ABB RAPID module: P2545L1ESegmentOrg.mod

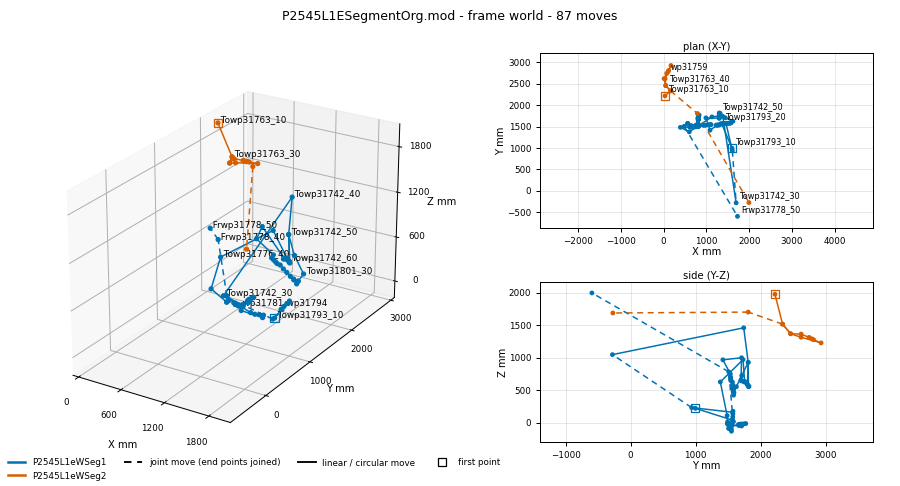
[picture p0: tool path of P2545L1ESegmentOrg.mod in frame world, 87 of 89 moves have a stored position in this frame; points joined in program order, loops and branches not executed]
%%%
  VERSION:1
  LANGUAGE:ENGLISH
%%%

MODULE P2545L1ESegment
!# Process Simulate on eMServer 14 to ABB Rapid Volvo download
!# ------------------------------------------------
!# CREATED   : 26/04/2018 14:09:44 by yogesha
!# CELL      : 2V3 Enginecase_V1
!# ROBOT     : AR21_IRB6700_220-265_SW_IRC5_Grey
!# PROGRAM   : P2545L1ESegment
!# VOLP      : Abb-Rapid-Volvo 3.14.1
!# RCS       : 6.04.irc5
!# CONTROLLER: 6.0 RW6


!# ----------------------------------------------
!# ------ ROBTARGET
!# ----------------------------------------------
  LOCAL CONST robtarget Towp31793_10:=[[4045.55,-245.18,1773.35],[0.031229,0.227881,0.973063,0.015622],[-1,0,-1,0],[9e+09,250,9e+09,9e+09,9e+09,9e+09]];
  LOCAL CONST robtarget Towp31793_20:=[[3464.22,18.06,1738.48],[0.0312267,0.227864,0.973067,0.0156211],[0,0,-1,0],[9E+09,250,9E+09,9E+09,9E+09,9E+09]];
  LOCAL CONST robtarget wp31793:=[[3459.52,28.59,1728.27],[0.0311732,0.227874,0.973066,0.0155927],[0,0,-1,0],[9E+09,24.9994,9E+09,9E+09,9E+09,9E+09]];
  LOCAL CONST robtarget wp31794:=[[3457.21,-31.09,1727.85],[0.0295957,0.184936,0.982299,0.00348625],[0,0,-1,0],[9E+09,25.0015,9E+09,9E+09,9E+09,9E+09]];
  LOCAL CONST robtarget wp31795:=[[3457.59,-92.13,1727.10],[0.0256679,0.112505,0.99332,0.000286719],[-1,1,-1,0],[9E+09,24.9989,9E+09,9E+09,9E+09,9E+09]];
  LOCAL CONST robtarget wp31796:=[[3459.26,-148.29,1728.07],[0.024545,0.091993,0.995457,-0.000992369],[-1,1,-1,0],[9E+09,24.9989,9E+09,9E+09,9E+09,9E+09]];
  LOCAL CONST robtarget Towp31742_10:=[[3464.44,-137.28,1737.71],[0.024542,0.091977,0.995458,-0.00102],[-1,1,-1,0],[9e+09,250,9e+09,9e+09,9e+09,9e+09]];
  LOCAL CONST robtarget Towp31742_20:=[[4102.65,-256.3,1769.61],[0.024542,0.091977,0.995458,-0.00102],[-1,0,-1,0],[9e+09,250,9e+09,9e+09,9e+09,9e+09]];
  LOCAL CONST robtarget Towp31742_30:=[[5323.84,-882.05,1248.86],[0.389563,-0.196475,-0.871387,-0.224327],[-1,0,-1,0],[9e+09,250,9e+09,9e+09,9e+09,9e+09]];
  LOCAL CONST robtarget Towp31742_40:=[[3288.74,-1093.58,858.48],[0.205443,-0.383752,-0.808886,-0.395262],[0,-1,0,0],[9E+09,200,9E+09,9E+09,9E+09,9E+09]];
  LOCAL CONST robtarget Towp31742_50:=[[3214.45,-634.81,1138.27],[0.192085,-0.483988,-0.79404,-0.313623],[0,-1,0,0],[9e+09,200,9e+09,9e+09,9e+09,9e+09]];
  LOCAL CONST robtarget Towp31742_60:=[[3228.3,-383.45,1373.91],[0.192085,-0.483988,-0.79404,-0.313623],[0,-1,0,0],[9e+09,200,9e+09,9e+09,9e+09,9e+09]];
  LOCAL CONST robtarget wp31742:=[[3218.38,-372.34,1363.36],[0.19209,-0.483981,-0.794042,-0.313625],[0,-1,0,0],[9E+09,25,9E+09,9E+09,9E+09,9E+09]];
  LOCAL CONST robtarget wp31743:=[[3202.14,-353.55,1377.18],[0.126687,-0.453575,-0.849352,-0.238374],[0,-1,0,0],[9E+09,25,9E+09,9E+09,9E+09,9E+09]];
  LOCAL CONST robtarget Towp31801_10:=[[3211.68,-359.85,1390.85],[0.126681,-0.453575,-0.849353,-0.238372],[0,-1,0,0],[9e+09,100,9e+09,9e+09,9e+09,9e+09]];
  LOCAL CONST robtarget Towp31801_20:=[[3214.45,-634.81,1138.27],[0.192085,-0.483988,-0.79404,-0.313623],[0,-1,0,0],[9e+09,200,9e+09,9e+09,9e+09,9e+09]];
  LOCAL CONST robtarget Towp31801_50:=[[3324.02,-564.37,1372.17],[0.253684,-0.525737,-0.694294,-0.420952],[0,-1,0,0],[9E+09,252.271,9E+09,9E+09,9E+09,9E+09]];
  LOCAL CONST robtarget Towp31801_30:=[[3418.53,-543.62,1612.1],[0.303641,-0.551478,-0.586786,-0.509271],[0,-1,1,0],[9e+09,300,9e+09,9e+09,9e+09,9e+09]];
  LOCAL CONST robtarget Towp31801_40:=[[3453.83,-438.28,1630.24],[0.30364,-0.551504,-0.586755,-0.509279],[0,-2,1,0],[9e+09,250,9e+09,9e+09,9e+09,9e+09]];
  LOCAL CONST robtarget wp31801:=[[3456.41,-397.01,1641.04],[0.303642,-0.551506,-0.586753,-0.509277],[0,-2,1,0],[9E+09,24.9995,9E+09,9E+09,9E+09,9E+09]];
  LOCAL CONST robtarget Towp31802_10:=[[3453.84,-438.28,1630.24],[0.30364,-0.551504,-0.586755,-0.509279],[0,-2,1,0],[9e+09,250,9e+09,9e+09,9e+09,9e+09]];
  LOCAL CONST robtarget Towp31802_20:=[[3460.41,-415.7,1573.72],[0.426749,-0.48377,-0.53862,-0.541977],[1,-2,1,0],[9e+09,250,9e+09,9e+09,9e+09,9e+09]];
  LOCAL CONST robtarget wp31802:=[[3457.06,-406.72,1584.59],[0.426746,-0.48378,-0.538616,-0.541976],[0,-2,1,0],[9E+09,25,9E+09,9E+09,9E+09,9E+09]];
  LOCAL CONST robtarget wp31803:=[[3459.02,-406.42,1523.09],[0.43668,-0.46746,-0.526416,-0.560069],[1,-2,1,0],[9E+09,25.0005,9E+09,9E+09,9E+09,9E+09]];
  LOCAL CONST robtarget wp31804:=[[3459.21,-407.58,1459.46],[0.445685,-0.447678,-0.547002,-0.549307],[1,-2,1,0],[9E+09,25,9E+09,9E+09,9E+09,9E+09]];
  LOCAL CONST robtarget wp31805:=[[3459.16,-405.57,1400.86],[0.452433,-0.455769,-0.540253,-0.543788],[1,-2,1,0],[9E+09,25,9E+09,9E+09,9E+09,9E+09]];
  LOCAL CONST robtarget wp31806:=[[3458.52,-409.86,1340.90],[0.439789,-0.439763,-0.5538,-0.553624],[1,-2,1,0],[9E+09,25,9E+09,9E+09,9E+09,9E+09]];
  LOCAL CONST robtarget wp400071:=[[3480.23,-407.44,1303.25],[0.415408,-0.44219,-0.578614,-0.545078],[1,-2,1,0],[9E+09,24.9993,9E+09,9E+09,9E+09,9E+09]];
  LOCAL CONST robtarget wp31807:=[[3480.96,-408.30,1277.13],[0.429146,-0.4291,-0.56212,-0.561897],[1,-2,1,0],[9E+09,25,9E+09,9E+09,9E+09,9E+09]];
  LOCAL CONST robtarget wp31808:=[[3479.48,-405.77,1244.18],[0.421356,-0.421308,-0.567923,-0.567823],[1,-2,1,0],[9E+09,25.0005,9E+09,9E+09,9E+09,9E+09]];
  LOCAL CONST robtarget wp31809:=[[3480.49,-404.93,1208.70],[0.421373,-0.421325,-0.56793,-0.56779],[1,-2,1,0],[9E+09,25,9E+09,9E+09,9E+09,9E+09]];
  LOCAL CONST robtarget Towp31738_10:=[[3484.07,-455.96,1198.82],[0.421374,-0.421319,-0.56794,-0.567784],[1,-2,1,0],[9e+09,200,9e+09,9e+09,9e+09,9e+09]];
  LOCAL CONST robtarget Towp31738_20:=[[3587.28,-510.98,927.08],[0.421374,-0.421319,-0.56794,-0.567784],[1,-2,1,0],[9e+09,200,9e+09,9e+09,9e+09,9e+09]];
  LOCAL CONST robtarget Towp31738_30:=[[3293.19,-486.33,848.58],[0.312249,-0.509804,-0.662688,-0.45105],[1,-1,1,0],[9E+09,100,9E+09,9E+09,9E+09,9E+09]];
  LOCAL CONST robtarget Towp31738_40:=[[3325.04,-426.92,1307.08],[0.481537,-0.548607,-0.510598,-0.454358],[1,-1,1,0],[9e+09,100,9e+09,9e+09,9e+09,9e+09]];
  LOCAL CONST robtarget wp31738:=[[3321.4,-408.44,1309.01],[0.481539,-0.548608,-0.510599,-0.454355],[1,-1,1,0],[9E+09,25,9E+09,9E+09,9E+09,9E+09]];
  LOCAL CONST robtarget wp31739:=[[3289.73,-404.44,1319.17],[0.411306,-0.529111,-0.571082,-0.474061],[1,-1,1,0],[9E+09,25,9E+09,9E+09,9E+09,9E+09]];
  LOCAL CONST robtarget wp31740:=[[3264.45,-398.53,1332.57],[0.350381,-0.565629,-0.615727,-0.42211],[0,-1,1,0],[9E+09,25,9E+09,9E+09,9E+09,9E+09]];
  LOCAL CONST robtarget Towp31776_10:=[[3270.4,-418.62,1333.94],[0.350381,-0.565628,-0.615725,-0.422114],[0,-1,1,0],[9e+09,100,9e+09,9e+09,9e+09,9e+09]];
  LOCAL CONST robtarget Towp31776_20:=[[3280.95,-555.22,975.55],[0.31225,-0.509807,-0.662682,-0.451053],[0,-1,1,0],[9e+09,200,9e+09,9e+09,9e+09,9e+09]];
  LOCAL CONST robtarget Towp31776_40:=[[3591.17,61.90,770.34],[0.307479,0.489827,-0.385208,0.719125],[1,-1,-1,0],[9E+09,200,9E+09,9E+09,9E+09,9E+09]];
  LOCAL CONST robtarget Towp31776_50:=[[3471.36,587.04,948.32],[0.504101,0.53927,-0.460831,0.492651],[1,-1,-1,0],[9E+09,200,9E+09,9E+09,9E+09,9E+09]];
  LOCAL CONST robtarget Towp31776_60:=[[3480,543.53,1199.86],[0.528139,0.542024,-0.467947,0.456404],[1,-1,-1,0],[9e+09,200,9e+09,9e+09,9e+09,9e+09]];
  LOCAL CONST robtarget wp31776:=[[3483.05,500.39,1205.78],[0.528141,0.542017,-0.46796,0.456396],[1,-1,-1,0],[9E+09,24.9917,9E+09,9E+09,9E+09,9E+09]];
  LOCAL CONST robtarget Towp31780_10:=[[3480,543.52,1199.86],[0.528138,0.542024,-0.467947,0.456404],[1,-1,-1,0],[9e+09,200,9e+09,9e+09,9e+09,9e+09]];
  LOCAL CONST robtarget Towp31780_20:=[[3390.65,544.94,1142.27],[0.528139,0.542024,-0.467946,0.456404],[1,-1,-1,0],[9e+09,200,9e+09,9e+09,9e+09,9e+09]];
  LOCAL CONST robtarget Towp31780_30:=[[3451.46,472,1330.74],[0.485437,0.649543,-0.468784,0.350265],[1,-1,-1,0],[9e+09,150,9e+09,9e+09,9e+09,9e+09]];
  LOCAL CONST robtarget wp31780:=[[3482.98,440.49,1321.01],[0.48544,0.649557,-0.468776,0.350246],[1,-1,-1,0],[9E+09,25,9E+09,9E+09,9E+09,9E+09]];
  LOCAL CONST robtarget wp31781:=[[3482.35,428.05,1352.01],[0.442766,0.654013,-0.507582,0.344363],[1,-1,-1,0],[9E+09,25.0005,9E+09,9E+09,9E+09,9E+09]];
  LOCAL CONST robtarget wp31785:=[[3464.69,396.47,1497.30],[0.470942,0.633397,-0.47932,0.383763],[1,-1,-1,0],[9E+09,25,9E+09,9E+09,9E+09,9E+09]];
  LOCAL CONST robtarget wp31786:=[[3461.70,368.27,1546.79],[0.379891,0.694641,-0.526925,0.309043],[1,-1,-1,0],[9E+09,25.0005,9E+09,9E+09,9E+09,9E+09]];
  LOCAL CONST robtarget wp31787:=[[3459.50,323.86,1589.21],[0.24633,0.70303,-0.621694,0.242006],[1,-1,-1,0],[9E+09,25.0005,9E+09,9E+09,9E+09,9E+09]];
  LOCAL CONST robtarget wp31788:=[[3459.95,282.60,1629.14],[0.353136,0.765889,-0.477535,0.246312],[1,-1,-1,0],[9E+09,24.9995,9E+09,9E+09,9E+09,9E+09]];
  LOCAL CONST robtarget Towp31782_10:=[[3455.66,320.67,1642.93],[0.353143,0.76587,-0.477559,0.246314],[1,-1,-1,0],[9e+09,100,9e+09,9e+09,9e+09,9e+09]];
  LOCAL CONST robtarget Towp31782_20:=[[3479.58,469.31,1398.3],[0.371118,0.727003,-0.513868,0.263966],[1,-1,-1,0],[9e+09,200,9e+09,9e+09,9e+09,9e+09]];
  LOCAL CONST robtarget wp31782:=[[3480.26,418.82,1363.79],[0.371131,0.726978,-0.513897,0.263958],[1,-1,-1,0],[9E+09,24.9974,9E+09,9E+09,9E+09,9E+09]];
  LOCAL CONST robtarget wp31775:=[[3460.80,422.79,1361.94],[0.369179,0.711005,-0.532671,0.272839],[1,-1,-1,0],[9E+09,24.9878,9E+09,9E+09,9E+09,9E+09]];
  LOCAL CONST robtarget wp31774:=[[3430.48,422.82,1360.70],[0.3679,0.715304,-0.528284,0.271855],[1,-1,-1,0],[9E+09,25,9E+09,9E+09,9E+09,9E+09]];
  LOCAL CONST robtarget Towp31767_10:=[[3431.36,435.91,1374.3],[0.36792,0.715269,-0.52832,0.271852],[1,-1,-1,0],[9e+09,75,9e+09,9e+09,9e+09,9e+09]];
  LOCAL CONST robtarget Towp31767_20:=[[3322.44,425.06,1380.62],[0.266606,0.650081,-0.667266,0.247126],[1,-1,-1,0],[9E+09,49.4176,9E+09,9E+09,9E+09,9E+09]];
  LOCAL CONST robtarget wp31767:=[[3217.64,388.64,1378.16],[0.161313,0.567008,-0.778505,0.21543],[1,-1,0,0],[9E+09,24.9979,9E+09,9E+09,9E+09,9E+09]];
  LOCAL CONST robtarget wp31768:=[[3241.82,402.64,1368.34],[0.265979,0.686435,-0.632244,0.241516],[1,-1,-1,0],[9E+09,25.0005,9E+09,9E+09,9E+09,9E+09]];
  LOCAL CONST robtarget wp31771:=[[3328.78,419.32,1363.33],[0.343843,0.752013,-0.470483,0.308051],[1,-1,-1,0],[9E+09,25,9E+09,9E+09,9E+09,9E+09]];
  LOCAL CONST robtarget wp31770:=[[3302.45,416.94,1357.38],[0.285253,0.752472,-0.498291,0.32268],[1,-1,-1,0],[9E+09,25,9E+09,9E+09,9E+09,9E+09]];
  LOCAL CONST robtarget wp31769:=[[3275.95,412.76,1358.82],[0.281989,0.697675,-0.612726,0.241452],[1,-1,-1,0],[9E+09,25,9E+09,9E+09,9E+09,9E+09]];
  LOCAL CONST robtarget Towp31779_10:=[[3279.73,435.49,1380.14],[0.281999,0.69766,-0.612741,0.241446],[1,-1,-1,0],[9e+09,75,9e+09,9e+09,9e+09,9e+09]];
  LOCAL CONST robtarget Towp31779_20:=[[3480.1,470.7,1295.95],[0.363356,0.754516,-0.492864,0.236144],[1,-1,-1,0],[9e+09,25,9e+09,9e+09,9e+09,9e+09]];
  LOCAL CONST robtarget wp31779:=[[3482.68,451.68,1288.55],[0.363388,0.754466,-0.492923,0.23613],[1,-1,-1,0],[9E+09,25,9E+09,9E+09,9E+09,9E+09]];
  LOCAL CONST robtarget wp31778:=[[3481.75,469.66,1267.37],[0.319477,0.752877,-0.529636,0.224937],[1,-1,-1,0],[9E+09,25.0005,9E+09,9E+09,9E+09,9E+09]];
  LOCAL CONST robtarget Frwp31778_10:=[[3480.1,470.71,1295.94],[0.363356,0.754516,-0.492864,0.236144],[1,-1,-1,0],[9e+09,75,9e+09,9e+09,9e+09,9e+09]];
  LOCAL CONST robtarget Frwp31778_20:=[[3451.42,471.98,1330.73],[0.550376,0.597256,-0.47701,0.335906],[1,-1,-1,0],[9E+09,75,9E+09,9E+09,9E+09,9E+09]];
  LOCAL CONST robtarget Frwp31778_30:=[[3390.65,544.94,1142.27],[0.528139,0.542024,-0.467946,0.456404],[1,-1,-1,0],[9e+09,100,9e+09,9e+09,9e+09,9e+09]];
  LOCAL CONST robtarget Frwp31778_40:=[[3452.82,11.54,588.04],[0.294229,0.459328,-0.391939,0.740831],[1,-1,-1,0],[9E+09,50,9E+09,9E+09,9E+09,9E+09]];
  LOCAL CONST robtarget Frwp31778_50:=[[6079.26,2565.85,1512.62],[0.516372,-0.844715,-0.107098,-0.091356],[0,-1,-2,0],[9e+09,50,9e+09,9e+09,9e+09,9e+09]];
  LOCAL CONST robtarget Towp31763_10:=[[3347.95,834.06,944.48],[0.127354,-0.51805,0.839702,0.101518],[0,0,-2,0],[9E+09,242,9E+09,9E+09,9E+09,9E+09]];
  LOCAL CONST robtarget Towp31763_30:=[[3426.57,520.60,1315.50],[0.184335,-0.578608,0.784931,-0.122949],[0,0,-2,0],[9E+09,242.273,9E+09,9E+09,9E+09,9E+09]];
  LOCAL CONST robtarget Towp31763_40:=[[3274.99,407.18,1434.32],[0.0363429,-0.545988,0.805467,-0.227595],[0,0,-2,0],[9E+09,242.273,9E+09,9E+09,9E+09,9E+09]];
  LOCAL CONST robtarget wp31763:=[[3171.50,283.07,1395.44],[6.03512E-05,0.582137,-0.813091,0.000137078],[1,0,-2,0],[9E+09,24.9948,9E+09,9E+09,9E+09,9E+09]];
  LOCAL CONST robtarget wp31759:=[[3176.67,136.97,1394.83],[0.0193566,-0.592124,0.805535,-0.0112687],[1,0,-2,0],[9E+09,24.9966,9E+09,9E+09,9E+09,9E+09]];
  LOCAL CONST robtarget wp31757:=[[3187.80,79.83,1395.86],[0.00985179,-0.606855,0.79473,-0.00582832],[1,0,-2,0],[9E+09,24.9978,9E+09,9E+09,9E+09,9E+09]];
  LOCAL CONST robtarget wp31756:=[[3187.98,48.79,1398.52],[8.77831E-06,0.626617,-0.779328,5.44794E-05],[1,-1,-2,0],[9E+09,25,9E+09,9E+09,9E+09,9E+09]];
  LOCAL CONST robtarget wp31752:=[[3189.26,-88.41,1398.85],[4.25555E-05,0.644101,-0.76494,0.000169744],[1,-1,-2,0],[9E+09,24.9996,9E+09,9E+09,9E+09,9E+09]];
  LOCAL CONST robtarget Frwp31752_10:=[[3195.54,257.28,1437.13],[0.0242655,-0.583135,0.797612,-0.152251],[0,0,-2,0],[9E+09,169.434,9E+09,9E+09,9E+09,9E+09]];
  LOCAL CONST robtarget Frwp31752_20:=[[3275.00,407.18,1434.32],[0.0363422,-0.54599,0.805466,-0.227593],[0,0,-2,0],[9E+09,242.273,9E+09,9E+09,9E+09,9E+09]];
  LOCAL CONST robtarget Frwp31752_30:=[[3426.57,520.60,1315.50],[0.184334,-0.578607,0.784932,-0.122949],[0,0,-2,0],[9E+09,242.273,9E+09,9E+09,9E+09,9E+09]];
  LOCAL CONST robtarget Frwp31752_50:=[[4215.11,789.08,1199.66],[0.410337,-0.682659,0.516184,-0.314887],[0,0,-2,0],[9e+09,10,9e+09,9e+09,9e+09,9e+09]];
  LOCAL CONST robtarget Frwp31752_60:=[[6189.98,2078.46,1654.43],[0.626282,-0.760131,-0.076663,-0.155225],[0,0,-2,0],[9e+09,10,9e+09,9e+09,9e+09,9e+09]];


!# -----------------------------------------------
!# ------ SPOT DATA
!# -----------------------------------------------
  LOCAL PERS spotdata Sd_wp31793:=[3179320,1,1,1,1,-1];
  LOCAL PERS spotdata Sd_wp31794:=[3179420,1,1,1,1,-1];
  LOCAL PERS spotdata Sd_wp31795:=[3179520,1,1,1,1,-1];
  LOCAL PERS spotdata Sd_wp31796:=[3179620,1,1,1,1,-1];
  LOCAL PERS spotdata Sd_wp31742:=[3174220,1,1,1,1,-1];
  LOCAL PERS spotdata Sd_wp31743:=[3174320,1,1,1,1,-1];
  LOCAL PERS spotdata Sd_wp31801:=[3180120,1,1,1,1,-1];
  LOCAL PERS spotdata Sd_wp31802:=[3180220,1,1,1,1,-1];
  LOCAL PERS spotdata Sd_wp31803:=[3180320,1,1,1,1,-1];
  LOCAL PERS spotdata Sd_wp31804:=[3180420,1,1,1,1,-1];
  LOCAL PERS spotdata Sd_wp31805:=[3180520,1,1,1,1,-1];
  LOCAL PERS spotdata Sd_wp31806:=[3180620,1,1,1,1,-1];
  LOCAL PERS spotdata Sd_wp400071:=[4007120,1,1,1,1,-1];
  LOCAL PERS spotdata Sd_wp31807:=[3180720,1,1,1,1,-1];
  LOCAL PERS spotdata Sd_wp31808:=[3180820,1,1,1,1,-1];
  LOCAL PERS spotdata Sd_wp31809:=[3180920,1,1,1,1,-1];
  LOCAL PERS spotdata Sd_wp31738:=[3173820,1,1,1,1,-1];
  LOCAL PERS spotdata Sd_wp31739:=[3173920,1,1,1,1,-1];
  LOCAL PERS spotdata Sd_wp31740:=[3174020,1,1,1,1,-1];
  LOCAL PERS spotdata Sd_wp31780:=[3178020,1,1,1,1,-1];
  LOCAL PERS spotdata Sd_wp31781:=[3178120,1,1,1,1,-1];
  LOCAL PERS spotdata Sd_wp31785:=[3178520,1,1,1,1,-1];
  LOCAL PERS spotdata Sd_wp31786:=[3178620,1,1,1,1,-1];
  LOCAL PERS spotdata Sd_wp31787:=[3178720,1,1,1,1,-1];
  LOCAL PERS spotdata Sd_wp31788:=[3178820,1,1,1,1,-1];
  LOCAL PERS spotdata Sd_wp31782:=[3178220,1,1,1,1,-1];
  LOCAL PERS spotdata Sd_wp31775:=[3177520,1,1,1,1,-1];
  LOCAL PERS spotdata Sd_wp31774:=[3177420,1,1,1,1,-1];
  LOCAL PERS spotdata Sd_wp31767:=[3176720,1,1,1,1,-1];
  LOCAL PERS spotdata Sd_wp31768:=[3176820,1,1,1,1,-1];
  LOCAL PERS spotdata Sd_wp31771:=[3177120,1,1,1,1,-1];
  LOCAL PERS spotdata Sd_wp31770:=[3177020,1,1,1,1,-1];
  LOCAL PERS spotdata Sd_wp31769:=[3176920,1,1,1,1,-1];
  LOCAL PERS spotdata Sd_wp31779:=[3177920,1,1,1,1,-1];
  LOCAL PERS spotdata Sd_wp31778:=[3177820,1,1,1,1,-1];
  LOCAL PERS spotdata Sd_wp31763:=[3176320,1,1,1,1,-1];
  LOCAL PERS spotdata Sd_wp31759:=[3175920,1,1,1,1,-1];
  LOCAL PERS spotdata Sd_wp31757:=[3175720,1,1,1,1,-1];
  LOCAL PERS spotdata Sd_wp31756:=[3175620,1,1,1,1,-1];
  LOCAL PERS spotdata Sd_wp31752:=[3175220,1,1,1,1,-1];
  LOCAL PERS spotdata Sd_wp31776:=[3177620,1,1,1,1,-1];

!# -----------------------------------------------
!# ------ WOBJ DATA
!# -----------------------------------------------
  PERS wobjdata wFM24_CabframeUQ53:=[FALSE,TRUE,"""",[[-210.08,4920.13,1168.24],[-0.310764,0.6630223,-0.6166411,0.2891035]],[[0,0,0],[1,0,0,0]]];
  PERS wobjdata wFM24_CabframeUQ54:=[FALSE,TRUE,"""",[[-212.9,4917.65,1167.66],[-0.3109636,0.6634134,-0.6162131,0.2889042]],[[0,0,0],[1,0,0,0]]];
  PERS wobjdata wFM24_Cabframe:=[FALSE,TRUE,"""",[[-210.08,4920.13,1168.24],[-0.310764,0.663022,-0.616641,0.289104]],[[0,0,0],[1,0,0,0]]];
  PERS wobjdata wFM24_CabframeGrip:=[FALSE,TRUE,"""",[[-2504.52,4649.77,2641.4],[0.1735002,0.9601499,-0.2131685,-0.0506865]],[[0,0,0],[1,0,0,0]]];




  PROC P2545L1eWSeg1()
     MoveAbsJ HomeXQ11Gun,v2500,fine,XQ11GunTCP;
     MoveL Towp31793_10,v2500,z200,XQ11GunTCP\Wobj:=wFM24_Cabframe;
     MoveL Towp31793_20,v2500,z50,XQ11GunTCP\Wobj:=wFM24_Cabframe;
     SpotL wp31793, v2500, XQ11Gun\GunD:=XQ11GunData, Sd_wp31793, XQ11GunTCP\WObj:=wFM24_Cabframe;
     SpotL wp31794, v2500, XQ11Gun\GunD:=XQ11GunData, Sd_wp31794, XQ11GunTCP\WObj:=wFM24_Cabframe;
     SpotL wp31795, v2500, XQ11Gun\GunD:=XQ11GunData, Sd_wp31795, XQ11GunTCP\WObj:=wFM24_Cabframe;
     SpotL wp31796, v2500, XQ11Gun\GunD:=XQ11GunData, Sd_wp31796, XQ11GunTCP\WObj:=wFM24_Cabframe;
     MoveL Towp31742_10,v2500,z200,XQ11GunTCP\Wobj:=wFM24_Cabframe;
     MoveL Towp31742_20,v2500,z200,XQ11GunTCP\Wobj:=wFM24_Cabframe;
     MoveJ Towp31742_30,v2500,z200,XQ11GunTCP\Wobj:=wFM24_Cabframe;
     MoveL Towp31742_40,v2500,z200,XQ11GunTCP\Wobj:=wFM24_Cabframe;
     MoveL Towp31742_50,v2500,z50,XQ11GunTCP\Wobj:=wFM24_Cabframe;
     MoveL Towp31742_60,v2500,z50,XQ11GunTCP\Wobj:=wFM24_Cabframe;
     SpotL wp31742, v2500, XQ11Gun\GunD:=XQ11GunData, Sd_wp31742, XQ11GunTCP\WObj:=wFM24_Cabframe;
     SpotL wp31743, v2500, XQ11Gun\GunD:=XQ11GunData, Sd_wp31743, XQ11GunTCP\WObj:=wFM24_Cabframe;
     MoveL Towp31801_10,v2500,z200,XQ11GunTCP\Wobj:=wFM24_Cabframe;
     MoveL Towp31801_20,v2500,z200,XQ11GunTCP\Wobj:=wFM24_Cabframe;
     MoveL Towp31801_50, v2500, z200, XQ11GunTCP\WObj:=wFM24_Cabframe;
     MoveL Towp31801_30,v2500,z50,XQ11GunTCP\Wobj:=wFM24_Cabframe;
     MoveL Towp31801_40,v2500,z50,XQ11GunTCP\Wobj:=wFM24_Cabframe;
     SpotL wp31801, v2500, XQ11Gun\GunD:=XQ11GunData, Sd_wp31801, XQ11GunTCP\WObj:=wFM24_Cabframe;
     MoveL Towp31802_10,v2500,z50,XQ11GunTCP\Wobj:=wFM24_Cabframe;
     MoveL Towp31802_20,v2500,z50,XQ11GunTCP\Wobj:=wFM24_Cabframe;
     SpotL wp31802, v2500, XQ11Gun\GunD:=XQ11GunData, Sd_wp31802, XQ11GunTCP\WObj:=wFM24_Cabframe;
     SpotL wp31803, v2500, XQ11Gun\GunD:=XQ11GunData, Sd_wp31803, XQ11GunTCP\WObj:=wFM24_Cabframe;
     SpotL wp31804, v2500, XQ11Gun\GunD:=XQ11GunData, Sd_wp31804, XQ11GunTCP\WObj:=wFM24_Cabframe;
     SpotL wp31805, v2500, XQ11Gun\GunD:=XQ11GunData, Sd_wp31805, XQ11GunTCP\WObj:=wFM24_Cabframe;
     SpotL wp31806, v2500, XQ11Gun\GunD:=XQ11GunData, Sd_wp31806, XQ11GunTCP\WObj:=wFM24_Cabframe;
     SpotL wp400071, v2500, XQ11Gun\GunD:=XQ11GunData, Sd_wp400071, XQ11GunTCP\WObj:=wFM24_Cabframe;
     SpotL wp31807, v2500, XQ11Gun\GunD:=XQ11GunData, Sd_wp31807, XQ11GunTCP\WObj:=wFM24_Cabframe;
     SpotL wp31808, v2500, XQ11Gun\GunD:=XQ11GunData, Sd_wp31808, XQ11GunTCP\WObj:=wFM24_Cabframe;
     SpotL wp31809, v2500, XQ11Gun\GunD:=XQ11GunData, Sd_wp31809, XQ11GunTCP\WObj:=wFM24_Cabframe;
     MoveL Towp31738_10,v2500,z50,XQ11GunTCP\Wobj:=wFM24_Cabframe;
     MoveL Towp31738_20,v2500,z50,XQ11GunTCP\Wobj:=wFM24_Cabframe;
     MoveL Towp31738_30,v2500,z50,XQ11GunTCP\Wobj:=wFM24_Cabframe;
     MoveL Towp31738_40,v2500,z50,XQ11GunTCP\Wobj:=wFM24_Cabframe;
     SpotL wp31738, v2500, XQ11Gun\GunD:=XQ11GunData, Sd_wp31738, XQ11GunTCP\WObj:=wFM24_Cabframe;
     SpotL wp31739, v2500, XQ11Gun\GunD:=XQ11GunData, Sd_wp31739, XQ11GunTCP\WObj:=wFM24_Cabframe;
     SpotL wp31740, v2500, XQ11Gun\GunD:=XQ11GunData, Sd_wp31740, XQ11GunTCP\WObj:=wFM24_Cabframe;
     MoveL Towp31776_10,v2500,z50,XQ11GunTCP\Wobj:=wFM24_Cabframe;
     MoveL Towp31776_20,v2500,z50,XQ11GunTCP\Wobj:=wFM24_Cabframe;
     MoveL Towp31776_40,v2500,z200,XQ11GunTCP\Wobj:=wFM24_Cabframe;
     MoveL Towp31776_50,v2500,z50,XQ11GunTCP\Wobj:=wFM24_Cabframe;
     MoveL Towp31776_60,v2500,z50,XQ11GunTCP\Wobj:=wFM24_Cabframe;
     SpotL wp31776, v2500, XQ11Gun\GunD:=XQ11GunData, Sd_wp31776, XQ11GunTCP\WObj:=wFM24_Cabframe;
     MoveL Towp31780_10,v2500,z50,XQ11GunTCP\Wobj:=wFM24_Cabframe;
     MoveL Towp31780_20,v2500,z50,XQ11GunTCP\Wobj:=wFM24_Cabframe;
     MoveL Towp31780_30,v2500,z50,XQ11GunTCP\Wobj:=wFM24_Cabframe;
     SpotL wp31780, v2500, XQ11Gun\GunD:=XQ11GunData, Sd_wp31780, XQ11GunTCP\WObj:=wFM24_Cabframe;
     SpotL wp31781, v2500, XQ11Gun\GunD:=XQ11GunData, Sd_wp31781, XQ11GunTCP\WObj:=wFM24_Cabframe;
     SpotL wp31785, v2500, XQ11Gun\GunD:=XQ11GunData, Sd_wp31785, XQ11GunTCP\WObj:=wFM24_Cabframe;
     SpotL wp31786, v2500, XQ11Gun\GunD:=XQ11GunData, Sd_wp31786, XQ11GunTCP\WObj:=wFM24_Cabframe;
     SpotL wp31787, v2500, XQ11Gun\GunD:=XQ11GunData, Sd_wp31787, XQ11GunTCP\WObj:=wFM24_Cabframe;
     SpotL wp31788, v2500, XQ11Gun\GunD:=XQ11GunData, Sd_wp31788, XQ11GunTCP\WObj:=wFM24_Cabframe;
     MoveL Towp31782_10,v2500,z50,XQ11GunTCP\Wobj:=wFM24_Cabframe;
     MoveL Towp31782_20,v2500,z50,XQ11GunTCP\Wobj:=wFM24_Cabframe;
     SpotL wp31782, v2500, XQ11Gun\GunD:=XQ11GunData, Sd_wp31782, XQ11GunTCP\WObj:=wFM24_Cabframe;
     SpotL wp31775, v2500, XQ11Gun\GunD:=XQ11GunData, Sd_wp31775, XQ11GunTCP\WObj:=wFM24_Cabframe;
     SpotL wp31774, v2500, XQ11Gun\GunD:=XQ11GunData, Sd_wp31774, XQ11GunTCP\WObj:=wFM24_Cabframe;
     MoveL Towp31767_10,v2500,z50,XQ11GunTCP\Wobj:=wFM24_Cabframe;
     MoveL Towp31767_20,v2500,z50,XQ11GunTCP\Wobj:=wFM24_Cabframe;
     SpotL wp31767, v2500, XQ11Gun\GunD:=XQ11GunData, Sd_wp31767, XQ11GunTCP\WObj:=wFM24_Cabframe;
     SpotL wp31768, v2500, XQ11Gun\GunD:=XQ11GunData, Sd_wp31768, XQ11GunTCP\WObj:=wFM24_Cabframe;
     SpotL wp31771,v2500,XQ11Gun\GunD:=XQ11GunData,Sd_wp31771,XQ11GunTCP\Wobj:=wFM24_Cabframe;
     SpotL wp31770,v2500,XQ11Gun\GunD:=XQ11GunData,Sd_wp31770,XQ11GunTCP\Wobj:=wFM24_Cabframe;
     SpotL wp31769,v2500,XQ11Gun\GunD:=XQ11GunData,Sd_wp31769,XQ11GunTCP\Wobj:=wFM24_Cabframe;
     MoveL Towp31779_10,v2500,z50,XQ11GunTCP\Wobj:=wFM24_Cabframe;
     MoveL Towp31779_20,v2500,z50,XQ11GunTCP\Wobj:=wFM24_Cabframe;
     SpotL wp31779,v2500,XQ11Gun\GunD:=XQ11GunData,Sd_wp31779,XQ11GunTCP\Wobj:=wFM24_Cabframe;
     SpotL wp31778,v2500,XQ11Gun\GunD:=XQ11GunData,Sd_wp31778,XQ11GunTCP\Wobj:=wFM24_Cabframe;
     MoveL Frwp31778_10,v2500,z50,XQ11GunTCP\Wobj:=wFM24_Cabframe;
     MoveL Frwp31778_20,v2500,z50,XQ11GunTCP\Wobj:=wFM24_Cabframe;
     MoveL Frwp31778_30,v2500,z200,XQ11GunTCP\Wobj:=wFM24_Cabframe;
     MoveJ Frwp31778_40,v2500,z200,XQ11GunTCP\Wobj:=wFM24_Cabframe;
     MoveJ Frwp31778_50, v2500, fine, XQ11GunTCP\WObj:=wFM24_CabframeGrip;
     RETURN;
  ENDPROC

  PROC P2545L1eWSeg2()
     MoveJ Towp31763_10,v2500,z200,XQ11GunTCP\Wobj:=wFM24_CabframeGrip;
     MoveL Towp31763_30,v2500,z200,XQ11GunTCP\Wobj:=wFM24_CabframeGrip;
     MoveL Towp31763_40,v2500,z50,XQ11GunTCP\Wobj:=wFM24_CabframeGrip;
     SpotL wp31763,v2500,XQ11Gun\GunD:=XQ11GunData,Sd_wp31763,XQ11GunTCP\Wobj:=wFM24_CabframeGrip;
     SpotL wp31759,v2500,XQ11Gun\GunD:=XQ11GunData,Sd_wp31759,XQ11GunTCP\Wobj:=wFM24_CabframeGrip;
     SpotL wp31757,v2500,XQ11Gun\GunD:=XQ11GunData,Sd_wp31757,XQ11GunTCP\Wobj:=wFM24_CabframeGrip;
     SpotL wp31756,v2500,XQ11Gun\GunD:=XQ11GunData,Sd_wp31756,XQ11GunTCP\Wobj:=wFM24_CabframeGrip;
     SpotL wp31752,v2500,XQ11Gun\GunD:=XQ11GunData,Sd_wp31752,XQ11GunTCP\Wobj:=wFM24_CabframeGrip;
     MoveL Frwp31752_10,v2500,z50,XQ11GunTCP\Wobj:=wFM24_CabframeGrip;
     MoveL Frwp31752_20,v2500,z200,XQ11GunTCP\Wobj:=wFM24_CabframeGrip;
     MoveL Frwp31752_30,v2500,z200,XQ11GunTCP\Wobj:=wFM24_CabframeGrip;
     MoveJ Frwp31752_50,v2500,z200,XQ11GunTCP\Wobj:=wFM24_CabframeGrip;
     MoveJ Frwp31752_60,v2500,z200,XQ11GunTCP\Wobj:=wFM24_CabframeGrip;
     MoveAbsJ HomeXQ11Gun,v2500,fine,XQ11GunTCP;
     RETURN;
  ENDPROC

ENDMODULE
